# EPICS substitutions: evrSupport/Db/ioc/IOC-LI21-MG01pattern.substitutions
#
# Pattern records
file evrPattern.template {
#	    Device        ,  SLC Pattern Check LNK    , EVR/Trigger
#	                                                  Links
  pattern { DEVICE        ,        LINK4              , LINK5 , LINK6 , LINKD }
	  { IOC:LI21:MG01 ,         ""                ,  ""   ,  ""   ,  ""   }
}
file evrPatternProc.template {
  pattern { DEVICE }
	  { IOC:LI21:MG01}
}
